PROGRAM MAIN
VAR
END_VAR

Manual();
Manual_1();

END_PROGRAM

(* stored: Version 1.1.0.1, ProductVersion 3.1.4024.6
   POU MAIN: Id {bebf08a9-dfaa-4c8e-987d-6b1ebeeda418}, SpecialFunc None *)
